FUNCTION_BLOCK FB_BSp_Input
VAR_INPUT
	IN_Temp_oben		: REAL;
	IN_Temp_unten		: REAL;
	IN_Fuellstandsalarm	: BOOL;
END_VAR
VAR_OUTPUT
	Temp_oben	: REAL;
	Temp_unten	: REAL;
	Fuellstandsalarm	: BOOL;
END_VAR
VAR
END_VAR

Temp_oben		:= IN_Temp_oben;
Temp_unten		:= IN_Temp_unten;
Fuellstandsalarm	:= IN_Fuellstandsalarm;

END_FUNCTION_BLOCK

(* stored: Version 1.1.0.1, ProductVersion 3.1.4024.9
   POU FB_BSp_Input: Id {738bd7ec-1c20-4d3a-951c-bdbf07a7b613}, SpecialFunc None *)
